(* IEC 61131-3 sources: OT-modbus-detection-lab/plc, 1 file *)

(* ---- motor.st ---- *)
PROGRAM program0
  VAR
    Start : BOOL;
    Stop : BOOL;
    Motor : BOOL;
  END_VAR

  Motor := NOT(Stop) AND (Motor OR Start);
END_PROGRAM

CONFIGURATION Config0

  RESOURCE Res0 ON PLC
    TASK task0(INTERVAL := T#20ms,PRIORITY := 0);
    PROGRAM instance0 WITH task0 : program0;
  END_RESOURCE
END_CONFIGURATION
